FUNCTION_BLOCK F_MUX_8 (* multiplexer *)
  (* Standard: 61131-3; Classification: standard selection function; Description: Copyright (c) 2013 TU Wien ACIN This program and the accompanying materials are made available under the terms of the Eclipse Public License 2.0 which is available at https://www.eclipse.org/legal/epl-2.0/ SPDX-License-Identifier: EPL-2.0 *)
  (* Version 1.0, 2026-05-29, Gemini CLI, 4diac-ide, created from F_MUX_4 *)
  PACKAGE iec61131::selection;
  {SET_ATTRIBUTE(eclipse4diac::core::GenericClassName, 'GEN_F_MUX')}
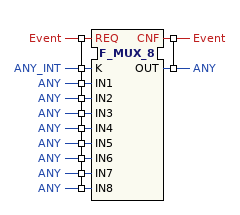
  EVENT_INPUT
    REQ WITH IN1, IN2, IN3, IN4, IN5, IN6, IN7, IN8, K; (* Service Request *)
  END_EVENT
  EVENT_OUTPUT
    CNF WITH OUT; (* Confirmation of Requested Service *)
  END_EVENT
  VAR_INPUT
    K : ANY_INT; (* Select one of n inputs *)
    IN1 : ANY; (* Input value 1 *)
    IN2 : ANY; (* Input value 2 *)
    IN3 : ANY; (* Input value 3 *)
    IN4 : ANY; (* Input value 4 *)
    IN5 : ANY; (* Input value 5 *)
    IN6 : ANY; (* Input value 6 *)
    IN7 : ANY; (* Input value 7 *)
    IN8 : ANY; (* Input value 8 *)
  END_VAR
  VAR_OUTPUT
    OUT : ANY; (* IN1 for K = 0, IN2 for K = 1, IN3 for K = 2, IN4 for K = 3, IN5 for K = 4, IN6 for K = 5, IN7 for K = 6, IN8 for K = 7 *)
  END_VAR
END_FUNCTION_BLOCK
